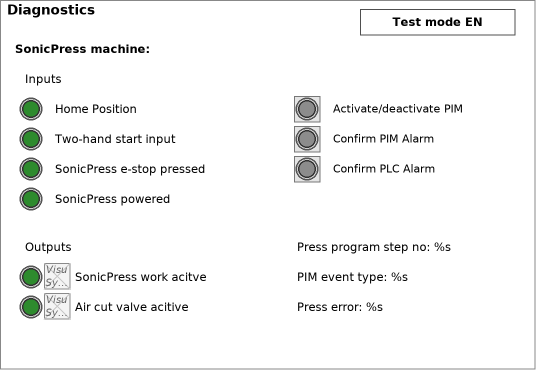
VISUALIZATION vSonicPress_SubDiag  // 536x370
VAR_IN_OUT
	fbMachine: fbSonicPress;
	fbPIM: fbPIM_Station_V3;
END_VAR
VAR
	bVisuTestMode: BOOL;
END_VAR
    Label (4,0 150x20), "Diagnostics"
    Label (12,36 203x26), "SonicPress machine:"
    Lamp1 (18,96 26x26), variable: fbMachine.stDigInOuts.bHomePosSensor, style: Lamp-Lamp1-Green
    Rectangle (52,96 160x26), "Home Position"
    Rectangle (52,126 160x26), "Two-hand start input"
    Lamp1 (18,126 26x26), variable: fbMachine.stDigInOuts.b2HandStart, style: Lamp-Lamp1-Green
    Lamp1 (18,156 26x26), variable: NOT fbMachine.stDigInOuts.bSafetyStatus, style: Lamp-Lamp1-Green
    Rectangle (52,156 160x26), "SonicPress e-stop pressed"
    Rectangle (22,66 160x26), "Inputs"
    Rectangle (22,234 160x26), "Outputs"
    Lamp1 (18,294 26x26), variable: fbMachine.stDigInOuts.bAirCutOffValve, style: Lamp-Lamp1-Green
    Lamp1 (18,264 26x26), variable: fbMachine.stDigInOuts.bPressGoDown_Q, style: Lamp-Lamp1-Green
    Rectangle (72,264 150x26), "SonicPress work acitve"
    Rectangle (72,294 150x26), "Air cut valve acitive"
    Rectangle (360,9 155x26), "Test mode EN", colour toggle: bVisuTestMode, input disabled if: NOT GVL.fbUserLogin.bPermissionGranted
        toggle fbMachine.bTestMode
        OnMouseClick: toggle bVisuTestMode
    Image (44,263 26x26), input disabled if: NOT bVisuTestMode, image: VisuSymbols.Symbols.Bracket
        OnMouseClick: toggle fbMachine.stDigInOuts.bPressGoDown_Q
    Image (44,293 26x26), input disabled if: NOT bVisuTestMode, image: VisuSymbols.Symbols.Bracket
        OnMouseClick: toggle fbMachine.stDigInOuts.bAirCutOffValve
    Lamp1 (18,186 26x26), variable: fbMachine.stDigInOuts.bPowerSupplyStatus, style: Lamp-Lamp1-Green
    Rectangle (52,186 160x26), "SonicPress powered"
    PushSwitch (294,96 26x26), variable: fbPIM.stPimInOut.bPIMActive, invisible if: Not bVisuTestMode, behaviour: TOGGLE, style: Switch-PushSwitch-Gray
    PushSwitch (294,126 26x26), variable: fbPIM.stPimInOut.bConfirmEvent, invisible if: Not bVisuTestMode, behaviour: TOGGLE, style: Switch-PushSwitch-Gray
    Label (330,96 150x26), "Activate/deactivate PIM", invisible if: Not bVisuTestMode
    Label (330,126 150x26), "Confirm PIM Alarm", invisible if: Not bVisuTestMode
    PushSwitch (294,156 26x26), variable: fbMachine.bServiceReset, invisible if: Not bVisuTestMode, behaviour: TOGGLE, style: Switch-PushSwitch-Gray
    Label (330,156 150x26), "Confirm PLC Alarm", invisible if: Not bVisuTestMode
    Rectangle (294,294 200x26), "Press error: %s", text variable: TO_STRING(fbMachine.nError), invisible if: NOT bVisuTestMode
    Rectangle (294,234 200x26), "Press program step no: %s", text variable: fbMachine.iWorkStep, invisible if: NOT bVisuTestMode
    Rectangle (294,264 200x26), "PIM event type: %s", text variable: TO_STRING(fbMachine.nEventActive), invisible if: NOT bVisuTestMode
END_VISUALIZATION

(* stored: Version 1.1.0.1, ProductVersion 3.1.4024.12
   Visu vSonicPress_SubDiag: Id {53e7843b-ac06-4fd0-b246-9f84d7e7d5c7} *)
